FUNCTION MINUTE : INT
VAR_INPUT
	itod : TOD;
END_VAR


(*
version 1.1	2 oct 2006
programmer 	hugo
tested by	tobias

extracts the minutes out of TOD truncating the seconds

*)

MINUTE := DWORD_TO_INT(TOD_TO_DWORD(itod) / 60000 - TOD_TO_DWORD(itod) / 3600000 * 60);


(* change history

2.10.2006 changes name of input to itod

*)

END_FUNCTION

(* stored: Version 1.1.0.1
   POU MINUTE: Id {b88e7e41-73c1-4b5d-9935-1cf159f404bb}, SpecialFunc None *)
